Yaskawa INFORM job: TCP_SHORT_SPIKE(FRONIUS)2.JBI

/JOB
//NAME TCP_SHORT_SPIKE(FRONIUS)2
///FOLDERNAME INNE
//POS
///NPOS 26,26,0,0,0,0
///TOOL 0
///POSTYPE PULSE
///PULSE
C00000=-4522,7890,92721,4183,103920,40722
C00001=51572,-18888,56851,3442,102879,51101
C00002=122982,-19772,56266,3351,102785,51058
C00003=159611,-22216,53415,3824,103992,41169
C00004=217908,-22431,53306,4360,103919,41358
C00005=-235462,-5269,75883,4614,104392,43838
C00006=-153545,-1072,81082,4849,103241,50558
C00007=-124293,-2636,78699,5089,105072,39210
C00008=-40227,-12346,65149,-3508,107000,-25624
C00009=-59133,-51472,18485,-3778,96982,-35770
C00010=-171218,-39835,31833,-3555,100205,-41270
C00011=-223636,-72206,121,-1301,90349,-10399
C00012=-33976,-100435,-18680,4384,67486,31782
C00013=35739,-70985,431,2854,84553,58647
C00014=-5678,-46953,23206,4094,98329,38645
C00015=-11803,-42926,27573,423,95273,79150
C00016=112606,-51089,19468,-1725,92616,88620
C00017=217978,-53301,17596,2620,92599,64894
C00018=-204884,-29921,43789,2305,99039,71251
C00019=-121309,-38471,33008,1392,96657,78068
C00020=760,-37860,33330,526,96785,77686
C00021=3014,-108295,-21684,521,54597,78361
C00022=-87172,-120926,-23399,-571,38876,88673
C00023=-215396,-111736,-22294,4322,52876,60061
C00024=118562,-111325,-22267,3244,53324,57850
C00025=194766,-104367,-19836,1977,59618,69494
BC00000=234604,127397,695026
BC00001=234605,127399,695029
BC00002=234605,127399,695029
BC00003=234605,127399,695029
BC00004=234605,127399,695029
BC00005=234604,127399,695026
BC00006=234605,127399,695029
BC00007=234605,127399,695029
BC00008=234605,127399,695029
BC00009=234605,127399,695029
BC00010=234605,127399,695029
BC00011=234605,127399,695029
BC00012=234605,127399,695029
BC00013=234605,127399,695027
BC00014=234605,127399,695029
BC00015=234605,127399,695026
BC00016=234605,127399,695026
BC00017=234605,127399,695026
BC00018=234605,127399,695024
BC00019=234605,127399,695026
BC00020=234605,127399,695026
BC00021=234605,127399,695026
BC00022=234605,127399,695026
BC00023=234605,127399,695026
BC00024=234605,127399,695026
BC00025=234605,127399,695026
//INST
///DATE 2023/10/04 15:16
///ATTR SC,RW
///GROUP1 RB1,BS1
NOP
MOVJ C00000 BC00000 VJ=0.78
MOVJ C00001 BC00001 VJ=0.78
MOVJ C00002 BC00002 VJ=0.78
MOVJ C00003 BC00003 VJ=0.78
MOVJ C00004 BC00004 VJ=0.78
MOVJ C00005 BC00005 VJ=0.78
MOVJ C00006 BC00006 VJ=0.78
MOVJ C00007 BC00007 VJ=0.78
MOVJ C00008 BC00008 VJ=0.78
MOVJ C00009 BC00009 VJ=0.78
MOVJ C00010 BC00010 VJ=0.78
MOVJ C00011 BC00011 VJ=0.78
MOVJ C00012 BC00012 VJ=0.78
MOVJ C00013 BC00013 VJ=0.78
MOVJ C00014 BC00014 VJ=0.78
'COMMENT
MOVJ C00015 BC00015 VJ=0.78
MOVJ C00016 BC00016 VJ=0.78
MOVJ C00017 BC00017 VJ=0.78
MOVJ C00018 BC00018 VJ=0.78
MOVJ C00019 BC00019 VJ=0.78
MOVJ C00020 BC00020 VJ=0.78
MOVJ C00021 BC00021 VJ=0.78
MOVJ C00022 BC00022 VJ=0.78
MOVJ C00023 BC00023 VJ=0.78
MOVJ C00024 BC00024 VJ=0.78
MOVJ C00025 BC00025 VJ=0.78
'COMMENT
END
